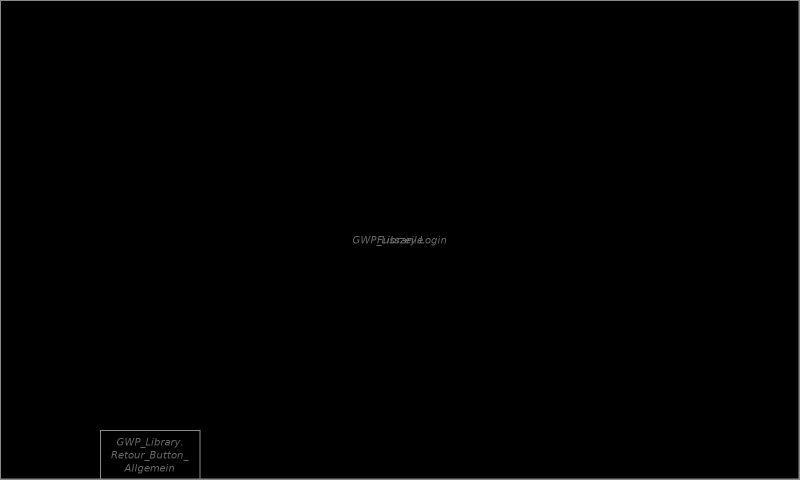
VISUALIZATION Login  // 800x480
    Frame (0,0 800x480)
        shows GWP_Library.Login()
    Frame (0,0 800x480)
        shows Fusszeile()
    Frame (100,430 100x50)
        shows GWP_Library.Retour_Button_Allgemein()
END_VISUALIZATION

(* stored: Version 1.1.0.1, ProductVersion 3.1.4022.6
   Visu Login: Id {ded1b158-d34a-4e09-9029-567708f5bde1} *)
